FUNCTION_BLOCK ABSTRACT CloneBase IMPLEMENTS ITF_Cloneable
VAR
END_VAR

METHOD ABSTRACT Clone : ITF_Cloneable
VAR_INPUT
END_VAR
END_METHOD

END_FUNCTION_BLOCK

(* stored: Version 1.1.0.1, ProductVersion 3.1.4024.12
   POU CloneBase: Id {213c3136-1102-4fd3-b410-62405f190958}, SpecialFunc None
   Method Clone: Id {619aaa26-bff4-4dd0-b018-2ad4c7fd4fa1} *)
